// TIA Portal V18 export
TYPE "Motor_Control"
   STRUCT
      Manual : Struct
         Start : Bool;
         CCWStart : Bool;
         SpeedChange : Bool;
      END_STRUCT;
      Auto : Struct
         Start : Bool;
         CCWStart : Bool;
         SpeedChange : Bool;
      END_STRUCT;
      OutControl : Struct
         o_Start : Bool;
         o_CCWStart : Bool;
         o_SpeedChanged : Bool;
         o_Ready : Bool;
         o_Alarm : Bool;
      END_STRUCT;
      Error : Array[0..15] of Bool;
   END_STRUCT;
   // // Error[0] : MotorControlDeviceAlarm
   // // Error[1] : PalletRunInTimeOut
   // // Error[2] : PalletRunOutTimeOut
END_TYPE
